// TwinCAT 3 PLC project PLC_Sim
// ProgramVersion: 3.1.4024.0
// libraries:
//   Tc2_Standard, * (Beckhoff Automation GmbH)
//   Tc2_System, * (Beckhoff Automation GmbH)
//   Tc3_Module, * (Beckhoff Automation GmbH)
// project tree:
//   / GlobalTextList.TcGTLO, PlcTask.TcTTO, Visualization Manager.TcVMO (not stored)
//   GVLs/ GVL.TcGVL
//   POUs/ MAIN.TcPOU, Process.TcPOU, Tramp.TcPOU
//   VISUs/ Visualization.TcVIS
// real-time tasks:
//   TASK PlcTask: cycle T#10ms, priority 20, ADS port 350
//   TASK PlcTask1: cycle T#10ms, priority 21, ADS port 351
// variable links:
//   PLC_Sim/PLC_Sim Instance <-> PLC_Student/PLC_Student Instance
//     PlcTask Inputs/GVL.ixDir <-> PlcTask Outputs/GVL.qxDir
//     PlcTask Inputs/GVL.ixStrobe <-> PlcTask Outputs/GVL.qxStrobe
//     PlcTask Outputs/GVL.qiAtStation1 <-> PlcTask Inputs/GVL.iiAtStation1
//     PlcTask Outputs/GVL.qiAtStation2 <-> PlcTask Inputs/GVL.iiAtStation2

CONFIGURATION PLC_Sim
    RESOURCE PLC ON TwinCAT3
        TASK PlcTask(INTERVAL := T#10ms, PRIORITY := 20);
        PROGRAM MAIN WITH PlcTask : MAIN;
    END_RESOURCE
END_CONFIGURATION

// ---- GVLs/GVL.TcGVL
{attribute 'qualified_only'}
VAR_GLOBAL
//Output from process to PLC
	ixStrobe		AT %I*:	BOOL;
	ixDir			AT %I*:	INT;
	
//Input to process from PLC
	qiAtStation1		AT %Q*:	BOOL;
	qiAtStation2		AT %Q*:	BOOL;
	qiDisplay		AT %Q*:	STRING;
END_VAR

// ---- POUs/MAIN.TcPOU
PROGRAM MAIN
VAR
END_VAR

Process();

END_PROGRAM

// ---- POUs/Process.TcPOU
PROGRAM Process
VAR
	Tramp_FB: Tramp;
END_VAR

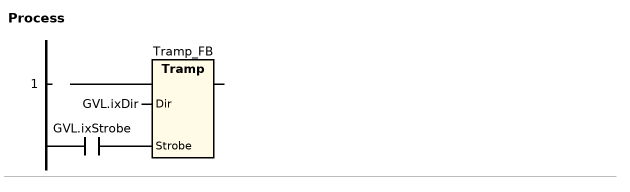
// NETWORK 1
Tramp_FB(Dir := GVL.ixDir, Strobe := GVL.ixStrobe); // Tramp

END_PROGRAM

// ---- POUs/Tramp.TcPOU
FUNCTION_BLOCK Tramp
VAR_INPUT
	Dir: INT := -1;
	Strobe: BOOL;
END_VAR
VAR_OUTPUT
END_VAR
VAR
	AtPos: INT;
	Goto_Pos: INT;
	Status: INT := 0;
	Error: BOOL;
	Speed: INT;
	Display : STRING;
END_VAR

IF Strobe THEN
	Goto_Pos := Goto_Pos + dir;
END_IF


GVL.qiAtStation1 := FALSE;
GVL.qiAtStation2 := FALSE;
IF AtPos > -50 AND atPos < 1 THEN
	GVL.qiAtStation1 := TRUE;
	//GVL.qiDisplay:='At Station1';
ELSIF AtPos > 550 AND atPos < 600 THEN
	GVL.qiAtStation2 := TRUE;
	//GVL.qiDisplay:='At Station2';
END_IF

IF AtPos > -40 AND AtPos <600 THEN
	AtPos := Goto_Pos;
	//GVL.qiDisplay:='On the way';
END_IF

END_FUNCTION_BLOCK

// ---- GlobalTextList.TcGTLO
TEXTLIST GlobalTextList
  834 = '%s'
  546 = 'AGV'
  253 = 'Error!'
  920 = 'S'
  533 = 'STATION -1'
  73 = 'STATION -2'
  381 = 'Station 1'
  873 = 'Station 2'
  2 = 'Station1'
  125 = 'Tram'
  507 = 'Tramp'
END_TEXTLIST

// ---- VISUs/Visualization.TcVIS
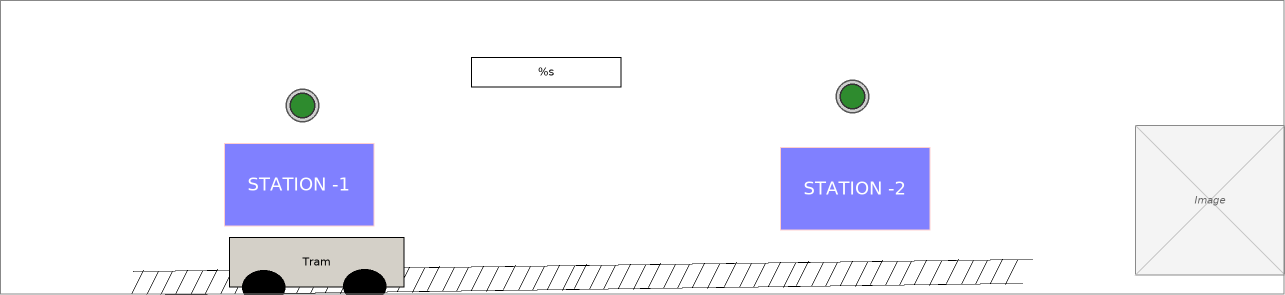
VISUALIZATION Visualization  // 1285x295
    Group (123,270 94x25)
        Line (0,25) (84,24)
        Line (20,0) (8,24)
        Line (35,1) (23,25)
        Line (49,1) (37,25)
        Line (64,0) (52,24)
        Line (79,1) (67,25)
        Line (10,1) (94,0)
    Group (197,269 94x25)
        Line (0,25) (84,24)
        Line (20,0) (8,24)
        Line (35,1) (23,25)
        Line (49,1) (37,25)
        Line (64,0) (52,24)
        Line (79,1) (67,25)
        Line (10,1) (94,0)
    Group (273,268 94x25)
        Line (0,25) (84,24)
        Line (20,0) (8,24)
        Line (35,1) (23,25)
        Line (49,1) (37,25)
        Line (64,0) (52,24)
        Line (79,1) (67,25)
        Line (10,1) (94,0)
    Group (345,267 94x25)
        Line (0,25) (84,24)
        Line (20,0) (8,24)
        Line (35,1) (23,25)
        Line (49,1) (37,25)
        Line (64,0) (52,24)
        Line (79,1) (67,25)
        Line (10,1) (94,0)
    Group (419,266 94x25)
        Line (0,25) (84,24)
        Line (20,0) (8,24)
        Line (35,1) (23,25)
        Line (49,1) (37,25)
        Line (64,0) (52,24)
        Line (79,1) (67,25)
        Line (10,1) (94,0)
    Group (495,265 94x25)
        Line (0,25) (84,24)
        Line (20,0) (8,24)
        Line (35,1) (23,25)
        Line (49,1) (37,25)
        Line (64,0) (52,24)
        Line (79,1) (67,25)
        Line (10,1) (94,0)
    Group (566,264 94x25)
        Line (0,25) (84,24)
        Line (20,0) (8,24)
        Line (35,1) (23,25)
        Line (49,1) (37,25)
        Line (64,0) (52,24)
        Line (79,1) (67,25)
        Line (10,1) (94,0)
    Group (640,263 94x25)
        Line (0,25) (84,24)
        Line (20,0) (8,24)
        Line (35,1) (23,25)
        Line (49,1) (37,25)
        Line (64,0) (52,24)
        Line (79,1) (67,25)
        Line (10,1) (94,0)
    Group (716,262 94x25)
        Line (0,25) (84,24)
        Line (20,0) (8,24)
        Line (35,1) (23,25)
        Line (49,1) (37,25)
        Line (64,0) (52,24)
        Line (79,1) (67,25)
        Line (10,1) (94,0)
    Group (788,261 94x25)
        Line (0,25) (84,24)
        Line (20,0) (8,24)
        Line (35,1) (23,25)
        Line (49,1) (37,25)
        Line (64,0) (52,24)
        Line (79,1) (67,25)
        Line (10,1) (94,0)
    Group (862,260 94x25)
        Line (0,25) (84,24)
        Line (20,0) (8,24)
        Line (35,1) (23,25)
        Line (49,1) (37,25)
        Line (64,0) (52,24)
        Line (79,1) (67,25)
        Line (10,1) (94,0)
    Group (938,259 94x25)
        Line (0,25) (84,24)
        Line (20,0) (8,24)
        Line (35,1) (23,25)
        Line (49,1) (37,25)
        Line (64,0) (52,24)
        Line (79,1) (67,25)
        Line (10,1) (94,0)
    Lamp1 (278,86 49x39), variable: GVL.qiAtStation1, style: Lamp-Lamp1-Green
    Lamp1 (828,77 49x39), variable: GVL.qiAtStation2, style: Lamp-Lamp1-Green
    Group (229,237 125x50)
        p3560616238: Process.Tramp_FB.AtPos
        RoundedRectangle (0,0 175x50), "Tram"
        Ellipse (13,33 43x34)
        Ellipse (114,32 43x34)
    Image (1135,125 150x150)
    RoundedRectangle (780,147 150x83), "STATION -2"
    RoundedRectangle (224,143 150x83), "STATION -1"
    Rectangle (471,57 150x30), "%s", text variable: GVL.qiDisplay
END_VISUALIZATION
